SUBAPPLICATION mapping_SFK (* Subapplication Type *)
  (* Standard: 61499-2 *)
  (* Version 1.0, 2023-02-07, franz *)
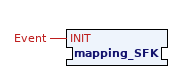
  EVENT_INPUT
    INIT;
  END_EVENT
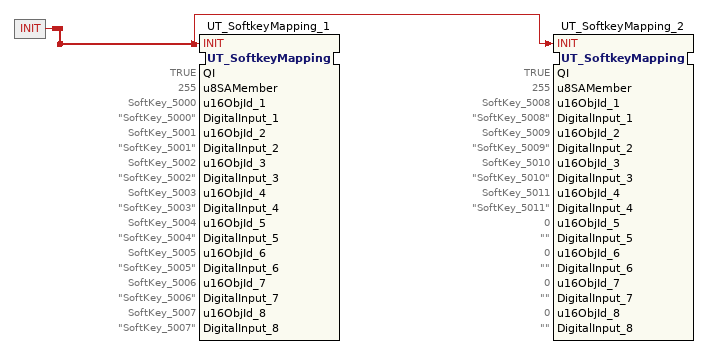
  FBS
    UT_SoftkeyMapping_1 : UT_SoftkeyMapping(QI := TRUE, u8SAMember := 255, u16ObjId_1 := SoftKey_5000, DigitalInput_1 := "SoftKey_5000", u16ObjId_2 := SoftKey_5001, DigitalInput_2 := "SoftKey_5001", u16ObjId_3 := SoftKey_5002, DigitalInput_3 := "SoftKey_5002", u16ObjId_4 := SoftKey_5003, DigitalInput_4 := "SoftKey_5003", u16ObjId_5 := SoftKey_5004, DigitalInput_5 := "SoftKey_5004", u16ObjId_6 := SoftKey_5005, DigitalInput_6 := "SoftKey_5005", u16ObjId_7 := SoftKey_5006, DigitalInput_7 := "SoftKey_5006", u16ObjId_8 := SoftKey_5007, DigitalInput_8 := "SoftKey_5007");
    UT_SoftkeyMapping_2 : UT_SoftkeyMapping(QI := TRUE, u8SAMember := 255, u16ObjId_1 := SoftKey_5008, DigitalInput_1 := "SoftKey_5008", u16ObjId_2 := SoftKey_5009, DigitalInput_2 := "SoftKey_5009", u16ObjId_3 := SoftKey_5010, DigitalInput_3 := "SoftKey_5010", u16ObjId_4 := SoftKey_5011, DigitalInput_4 := "SoftKey_5011", u16ObjId_5 := 0, DigitalInput_5 := "", u16ObjId_6 := 0, DigitalInput_6 := "", u16ObjId_7 := 0, DigitalInput_7 := "", u16ObjId_8 := 0, DigitalInput_8 := "");
  END_FBS
  EVENT_CONNECTIONS
    INIT TO UT_SoftkeyMapping_1.INIT;
    INIT TO UT_SoftkeyMapping_2.INIT;
  END_CONNECTIONS
END_SUBAPPLICATION
